// TIA Portal V17 export
// export: Created 2023-03-28T14:06:50.8846971Z, ExportSetting WithDefaults, DisplayName Totally Integrated Automation Portal, DisplayVersion V17 Update 4, DisplayName TIA Portal Openness, DisplayVersion V17 Update 4, DisplayName TIA Portal Version Control Interface, DisplayVersion V17, DisplayName STEP 7 Professional, DisplayVersion V17 Update 4, DisplayName STEP 7 Safety, DisplayVersion V17, DisplayName WinCC Professional, DisplayVersion V17 Update 4
FUNCTION "PCS1 R (S)" : Void   // FC43, LAD
TITLE = ModBus TCP for PCS Power Electronics
{ S7_Optimized_Access := 'TRUE' }
VERSION : 0.1
// stored: AutoNumber false, IsIECCheckEnabled false, SetENOAutomatically false, UDAEnableTagReadback false
   VAR_TEMP
      rVac : Real;
   END_VAR
   VAR_TEMP   // added for the SCL form of the ladder/FBD networks
      _w1 : Bool;
   END_VAR
BEGIN

REGION Network 1: Function Modbus Client
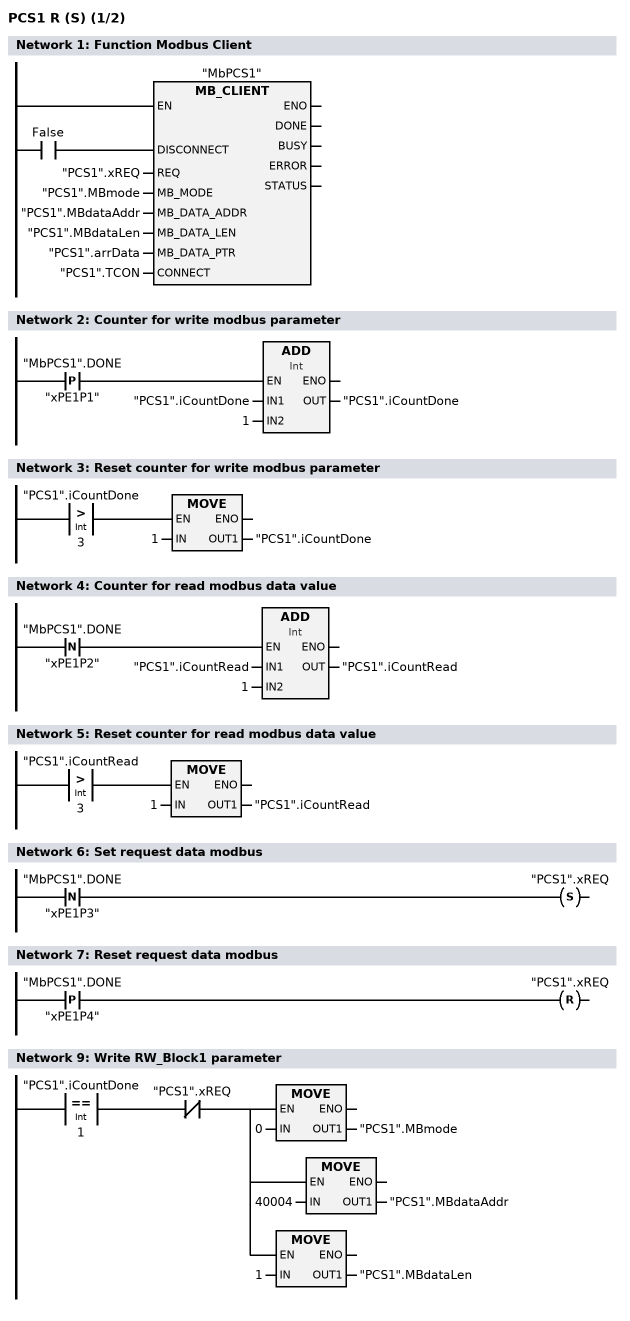
   RUNG wire#powerrail
      "MbPCS1".MB_CLIENT(DISCONNECT := wire#w1, REQ := "PCS1".xREQ, MB_MODE := "PCS1".MBmode, MB_DATA_ADDR := "PCS1".MBdataAddr, MB_DATA_LEN := "PCS1".MBdataLen, MB_DATA_PTR := "PCS1".arrData, CONNECT := "PCS1".TCON, DONE =>, BUSY =>, ERROR =>, STATUS =>)
   END_RUNG
   RUNG wire#powerrail
      Contact( False )
   END_RUNG wire#w1
   // the same network as SCL:
   "MbPCS1"(DISCONNECT := False,   // MB_CLIENT
            REQ := "PCS1".xREQ,
            MB_MODE := "PCS1".MBmode,
            MB_DATA_ADDR := "PCS1".MBdataAddr,
            MB_DATA_LEN := "PCS1".MBdataLen,
            MB_DATA_PTR := "PCS1".arrData,
            CONNECT := "PCS1".TCON);
END_REGION

REGION Network 2: Counter for write modbus parameter
   RUNG wire#powerrail
      P_Contact(operand := "MbPCS1".DONE, bit := "xPE1P1")
      { S7_Templates := "SrcType := Int" } Add(in1 := "PCS1".iCountDone, in2 := 1, out => "PCS1".iCountDone)
   END_RUNG
   // the same network as SCL:
   #_w1 := "MbPCS1".DONE AND NOT "xPE1P1";   // rising edge of "MbPCS1".DONE
   "xPE1P1" := "MbPCS1".DONE;
   IF #_w1 THEN "PCS1".iCountDone := "PCS1".iCountDone + 1; END_IF;
END_REGION

REGION Network 3: Reset counter for write modbus parameter
   RUNG wire#powerrail
      { S7_Templates := "SrcType := Int" } GT_Contact(in1 := "PCS1".iCountDone, in2 := 3)
      Move(in := 1, out1 => "PCS1".iCountDone)
   END_RUNG
   // the same network as SCL:
   IF "PCS1".iCountDone > 3 THEN "PCS1".iCountDone := 1; END_IF;
END_REGION

REGION Network 4: Counter for read modbus data value
   RUNG wire#powerrail
      N_Contact(operand := "MbPCS1".DONE, bit := "xPE1P2")
      { S7_Templates := "SrcType := Int" } Add(in1 := "PCS1".iCountRead, in2 := 1, out => "PCS1".iCountRead)
   END_RUNG
   // the same network as SCL:
   #_w1 := NOT "MbPCS1".DONE AND "xPE1P2";   // falling edge of "MbPCS1".DONE
   "xPE1P2" := "MbPCS1".DONE;
   IF #_w1 THEN "PCS1".iCountRead := "PCS1".iCountRead + 1; END_IF;
END_REGION

REGION Network 5: Reset counter for read modbus data value
   RUNG wire#powerrail
      { S7_Templates := "SrcType := Int" } GT_Contact(in1 := "PCS1".iCountRead, in2 := 3)
      Move(in := 1, out1 => "PCS1".iCountRead)
   END_RUNG
   // the same network as SCL:
   IF "PCS1".iCountRead > 3 THEN "PCS1".iCountRead := 1; END_IF;
END_REGION

REGION Network 6: Set request data modbus
   RUNG wire#powerrail
      N_Contact(operand := "MbPCS1".DONE, bit := "xPE1P3")
      S_Coil( "PCS1".xREQ )
   END_RUNG
   // the same network as SCL:
   #_w1 := NOT "MbPCS1".DONE AND "xPE1P3";   // falling edge of "MbPCS1".DONE
   "xPE1P3" := "MbPCS1".DONE;
   IF #_w1 THEN "PCS1".xREQ := TRUE; END_IF;
END_REGION

REGION Network 7: Reset request data modbus
   RUNG wire#powerrail
      P_Contact(operand := "MbPCS1".DONE, bit := "xPE1P4")
      R_Coil( "PCS1".xREQ )
   END_RUNG
   // the same network as SCL:
   #_w1 := "MbPCS1".DONE AND NOT "xPE1P4";   // rising edge of "MbPCS1".DONE
   "xPE1P4" := "MbPCS1".DONE;
   IF #_w1 THEN "PCS1".xREQ := FALSE; END_IF;
END_REGION

REGION Network 9: Write RW_Block1 parameter
   RUNG wire#powerrail
      { S7_Templates := "SrcType := Int" } EQ_Contact(in1 := "PCS1".iCountDone, in2 := 1)
      I_Contact( "PCS1".xREQ )
      wire#w1
      Move(in := 0, out1 => "PCS1".MBmode)
   END_RUNG
   RUNG wire#w1
      Move(in := 40004, out1 => "PCS1".MBdataAddr)
   END_RUNG
   RUNG wire#w1
      Move(in := 1, out1 => "PCS1".MBdataLen)
   END_RUNG
   // the same network as SCL:
   IF ("PCS1".iCountDone = 1) AND NOT "PCS1".xREQ THEN
       "PCS1".MBmode := 0;
       "PCS1".MBdataAddr := 40004;
       "PCS1".MBdataLen := 1;
   END_IF;
END_REGION

REGION Network 10: Read RW_Block1 data value
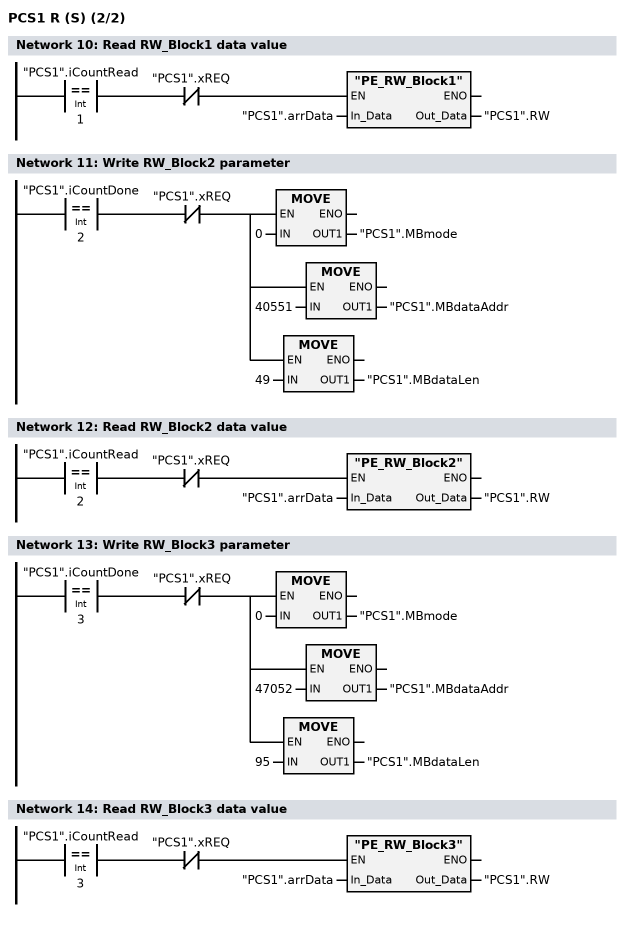
   RUNG wire#powerrail
      { S7_Templates := "SrcType := Int" } EQ_Contact(in1 := "PCS1".iCountRead, in2 := 1)
      I_Contact( "PCS1".xREQ )
      "PE_RW_Block1"(In_Data := "PCS1".arrData, Out_Data => "PCS1".RW)
   END_RUNG
   // the same network as SCL:
   IF ("PCS1".iCountRead = 1) AND NOT "PCS1".xREQ THEN
       "PE_RW_Block1"(In_Data := "PCS1".arrData, Out_Data => "PCS1".RW);
   END_IF;
END_REGION

REGION Network 11: Write RW_Block2 parameter
   RUNG wire#powerrail
      { S7_Templates := "SrcType := Int" } EQ_Contact(in1 := "PCS1".iCountDone, in2 := 2)
      I_Contact( "PCS1".xREQ )
      wire#w1
      Move(in := 0, out1 => "PCS1".MBmode)
   END_RUNG
   RUNG wire#w1
      Move(in := 40551, out1 => "PCS1".MBdataAddr)
   END_RUNG
   RUNG wire#w1
      Move(in := 49, out1 => "PCS1".MBdataLen)
   END_RUNG
   // the same network as SCL:
   IF ("PCS1".iCountDone = 2) AND NOT "PCS1".xREQ THEN
       "PCS1".MBmode := 0;
       "PCS1".MBdataAddr := 40551;
       "PCS1".MBdataLen := 49;
   END_IF;
END_REGION

REGION Network 12: Read RW_Block2 data value
   RUNG wire#powerrail
      { S7_Templates := "SrcType := Int" } EQ_Contact(in1 := "PCS1".iCountRead, in2 := 2)
      I_Contact( "PCS1".xREQ )
      "PE_RW_Block2"(In_Data := "PCS1".arrData, Out_Data => "PCS1".RW)
   END_RUNG
   // the same network as SCL:
   IF ("PCS1".iCountRead = 2) AND NOT "PCS1".xREQ THEN
       "PE_RW_Block2"(In_Data := "PCS1".arrData, Out_Data => "PCS1".RW);
   END_IF;
END_REGION

REGION Network 13: Write RW_Block3 parameter
   RUNG wire#powerrail
      { S7_Templates := "SrcType := Int" } EQ_Contact(in1 := "PCS1".iCountDone, in2 := 3)
      I_Contact( "PCS1".xREQ )
      wire#w1
      Move(in := 0, out1 => "PCS1".MBmode)
   END_RUNG
   RUNG wire#w1
      Move(in := 47052, out1 => "PCS1".MBdataAddr)
   END_RUNG
   RUNG wire#w1
      Move(in := 95, out1 => "PCS1".MBdataLen)
   END_RUNG
   // the same network as SCL:
   IF ("PCS1".iCountDone = 3) AND NOT "PCS1".xREQ THEN
       "PCS1".MBmode := 0;
       "PCS1".MBdataAddr := 47052;
       "PCS1".MBdataLen := 95;
   END_IF;
END_REGION

REGION Network 14: Read RW_Block3 data value
   RUNG wire#powerrail
      { S7_Templates := "SrcType := Int" } EQ_Contact(in1 := "PCS1".iCountRead, in2 := 3)
      I_Contact( "PCS1".xREQ )
      "PE_RW_Block3"(In_Data := "PCS1".arrData, Out_Data => "PCS1".RW)
   END_RUNG
   // the same network as SCL:
   IF ("PCS1".iCountRead = 3) AND NOT "PCS1".xREQ THEN
       "PE_RW_Block3"(In_Data := "PCS1".arrData, Out_Data => "PCS1".RW);
   END_IF;
END_REGION
END_FUNCTION
